PROGRAM P_AdsLicenseServer
VAR
    fbWriteInd  : ADSWRITEIND;
    fbWriteRes  : ADSWRITERES;

    fbReadInd   : ADSREADIND;
    fbReadRes   : ADSREADRES;

    bClearWrite : BOOL := FALSE;
    bClearRead  : BOOL := FALSE;

    pWriteData  : POINTER TO STRING(80);
    sProductId  : STRING(80);

    sTrialToken : STRING(256) := 'NO_LICENSE';

    cIG_RequestTrial  : UDINT := 16#80000001; // must have MSB = 1
    cIG_GetTrialToken : UDINT := 16#80000002;
END_VAR

// --- HANDLE WRITE (request) ---
fbWriteInd(CLEAR := bClearWrite);
bClearWrite := FALSE;

IF fbWriteInd.VALID THEN
    IF fbWriteInd.IDXGRP = cIG_RequestTrial THEN
        pWriteData := fbWriteInd.DATAADDR;
        sProductId := pWriteData^; // assume it's null-terminated STRING

        sTrialToken := CONCAT('TRIAL_', sProductId); 
        sTrialToken := CONCAT(sTrialToken, '_OK');

        fbWriteRes(
            NETID    := fbWriteInd.NETID,
            PORT     := fbWriteInd.PORT,
            INVOKEID := fbWriteInd.INVOKEID,
            RESULT   := 0,
            RESPOND  := TRUE
        );
    ELSE
        fbWriteRes(
            NETID    := fbWriteInd.NETID,
            PORT     := fbWriteInd.PORT,
            INVOKEID := fbWriteInd.INVOKEID,
            RESULT   := 16#701,
            RESPOND  := TRUE
        );
    END_IF
    bClearWrite := TRUE;
END_IF

// --- HANDLE READ (client wants token) ---
fbReadInd(CLEAR := bClearRead);
bClearRead := FALSE;

IF fbReadInd.VALID THEN
    IF fbReadInd.IDXGRP = cIG_GetTrialToken THEN
        fbReadRes(
            NETID    := fbReadInd.NETID,
            PORT     := fbReadInd.PORT,
            INVOKEID := fbReadInd.INVOKEID,
            RESULT   := 0,
            LEN      := SIZEOF(sTrialToken),
            DATAADDR := ADR(sTrialToken),
            RESPOND  := TRUE
        );
    ELSE
        fbReadRes(
            NETID    := fbReadInd.NETID,
            PORT     := fbReadInd.PORT,
            INVOKEID := fbReadInd.INVOKEID,
            RESULT   := 16#701,
            LEN      := 0,
            DATAADDR := 0,
            RESPOND  := TRUE
        );
    END_IF
    bClearRead := TRUE;
END_IF

END_PROGRAM

(* stored: Version 1.2.0.0, ProductVersion 3.1.4026.13, FileIdentifier 75b3a4b7b3b44fc6c30c0a484609380e128c4d83, FileSignature 6568aeed8c16ce7f404428ae0e7b4cc660140cb3b54c319e2d1685b59c6b9c6da3157259cacdb99ee2302b5a47a9fe7c51d75408660f43266a0334e1a4a3045a8930fb1e0eeae686ce8bfe3af61596fb99853def7988b106e47e0c1124da58f7962b2199190103c60e12aada55287a3496ac46c5691ae8699d6c49b3ca3815e17fae6a0b25d2fc2eed65e5d20af8f6fcb1a2a65587bee9a7a1909b07d20aa85ba81fe0484e155096708a78119459894aa562217a33a1223e400a73884ed8b66b278e3d8065fe9c21a72ae794e8e6d980bac54fc371f8d747eea5007baa3db509cbb0894cbb8e98382df2cdbbcd1426e24cb5777f4e986c1a1b9fa727b04e7934
   POU P_AdsLicenseServer: Id {d02e1468-d291-47d8-9b1c-924fc194640c}, SpecialFunc None *)
